Staubli VAL3: ex11.dtx

jointRx jdepart = {j1=134.407099, j2=26.523821, j3=33.675048, j4=-3.327828, j5=91.404305, j6=185.663158}
mdesc mNomSpeed
mdesc mlent = {accel=9, vel=30, decel=9, blend=off}
pointRx ppa = {x=-389.287784, y=53.146528, z=-28.653819, rx=3.121688, ry=179.928998, rz=43.138261, fatherId=world[0]}
pointRx ppb = {x=-392.751036, y=2.592415, z=-1.732499, rx=3.435817, ry=-175.972362, rz=35.966227, fatherId=world[0]}
pointRx ppc = {x=-443.813598, y=21.968017, z=-61.84437, rx=4.174068, ry=-171.391146, rz=38.207024, fatherId=world[0]}
pointRx ppd = {x=-421.04634, y=36.124755, z=-39.679222, rx=3.922497, ry=-175.031609, rz=40.248351, fatherId=world[0]}
pointRx ppe = {x=-448.066006, y=58.834313, z=21.091808, rx=3.194213, ry=-168.378902, rz=44.251398, fatherId=world[0]}
pointRx ppf = {x=-436.387446, y=117.43347, z=21.091808, rx=4.715867, ry=-168.902608, rz=36.413108, fatherId=world[0]}
pointRx ppg = {x=-376.501098, y=118.984044, z=90.989667, rx=3.551758, ry=-174.364682, rz=22.207377, fatherId=world[0]}
tool tstylo = {z=180, fatherId=flange[0], ioLink=valve1}
